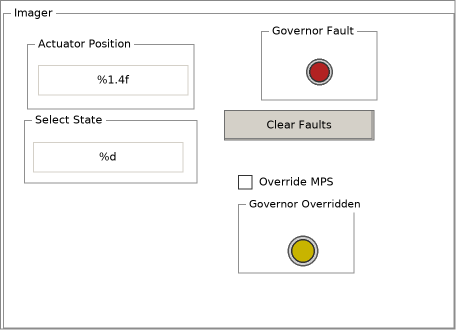
VISUALIZATION ImagerGUI  // 456x330
VAR_IN_OUT
	stDevice	:	ST_Device;
	fbDevice	:	FB_ExampleDeviceSM_All;
END_VAR
    GroupBox (3,5 451x323), "Imager"
        Button (221,105 150x30), "Clear Faults", pressed state: stDevice.xClearFaults
            tap stDevice.xClearFaults
        Checkbox (233,162 150x30), "Override MPS"
        GroupBox (258,18 116x77), "Governor Fault"
            Lamp1 (43,33 31x32), variable: stDevice.xGovernorFault, style: Lamp-Lamp1-Red
        GroupBox (235,191 116x77), "Governor Overridden"
            Lamp1 (47,35 36x40), variable: stDevice.xGovernorOverridden, style: Lamp-Lamp1-Yellow
        GroupBox (24,31 167x73), "Actuator Position"
            Textfield (11,29 150x30), "%1.4f", text variable: stDevice.stAxis.NcToPlc.ActPos
        GroupBox (21,107 173x71), "Select State"
            Textfield (9,30 150x30), "%d", text variable: stDevice.nRequestedState
                OnMouseDown: write the text variable via Default
END_VISUALIZATION

(* stored: Version 1.1.0.1, ProductVersion 3.1.4022.18
   Visu ImagerGUI: Id {c4e9eed9-0847-0b0c-1a64-5b138d22d3b0} *)
